(*			
	EVERDE sp. z o.o.
	Rafał Osajda		31.01.2025		TC 4026.13		wer. 0.0.0.1
	Obsługa przycisków 
*)
FUNCTION_BLOCK ABSTRACT FB_Button EXTENDS FB_BaseComponent IMPLEMENTS ITF_Button
VAR
	bContact							AT %I*	: BOOL;		// Styk przycisku 
	bContactPrev								: BOOL;
END_VAR

METHOD PUBLIC GetRisingEdgePressed : BOOL
VAR_INPUT
END_VAR
END_METHOD

(*			
	EVERDE sp. z o.o.
	Rafał Osajda		31.01.2025		TC 4026.13		wer. 0.0.0.1
	Zwraca stan przycisku
*)
METHOD IsPressed : BOOL
END_METHOD

END_FUNCTION_BLOCK

(* stored: Version 1.1.0.1
   POU FB_Button: Id {85c8c0af-9b54-4c45-a5dc-25d08c07092f}, SpecialFunc None
   Method GetRisingEdgePressed: Id {660354d3-961d-0c50-2f7c-6ceb634fdf0d}
   Method IsPressed: Id {c057585d-3d71-4e42-ba48-ae55c4f30095} *)
